   cmMendrelCathodeFrontClamp.configuration.disableFeedbackHomePos := FALSE;
   cmMendrelCathodeFrontClamp.configuration.disableFeedbackWorkPos := FALSE;
   cmMendrelCathodeFrontClamp.configuration.disableAlarms := FALSE;
   cmMendrelCathodeFrontClamp.configuration.resetOutputsOnError := FALSE;
   cmMendrelCathodeFrontClamp.configuration.allwaysWaitOnReachingTime := FALSE;
   cmMendrelCathodeRearClamp.commands.refreshConfiguration := FALSE;
   cmMendrelCathodeRearClamp.commands.editConfiguration := FALSE;
   cmMendrelCathodeRearClamp.commands.saveConfiguration := FALSE;
   cmMendrelCathodeRearClamp.commands.reset := FALSE;
   cmMendrelCathodeRearClamp.commands.commandHomePos := FALSE;
   cmMendrelCathodeRearClamp.commands.commandWorkPos := FALSE;
   cmMendrelCathodeRearClamp.monitoring.enable := TRUE;
   cmMendrelCathodeRearClamp.monitoring.referenceDesignator := WSTRING#'MendrelCathodeRearClamp';
   cmMendrelCathodeRearClamp.monitoring.commandHomePos := FALSE;
   cmMendrelCathodeRearClamp.monitoring.commandWorkPos := FALSE;
   cmMendrelCathodeRearClamp.monitoring.goToHomePos := FALSE;
   cmMendrelCathodeRearClamp.monitoring.goToWorkPos := TRUE;
   cmMendrelCathodeRearClamp.monitoring.inHomePos := FALSE;
   cmMendrelCathodeRearClamp.monitoring.inWorkPos := TRUE;
   cmMendrelCathodeRearClamp.monitoring.reset := FALSE;
   cmMendrelCathodeRearClamp.monitoring.enableManualCmds := FALSE;
   cmMendrelCathodeRearClamp.monitoring.error := FALSE;
   cmMendrelCathodeRearClamp.monitoring.interlockHomePos := TRUE;
   cmMendrelCathodeRearClamp.monitoring.interlockWorkPos := TRUE;
   cmMendrelCathodeRearClamp.monitoring.status := 16#7006;
   cmMendrelCathodeRearClamp.monitoring.interlockWarningWorkPos := FALSE;
   cmMendrelCathodeRearClamp.monitoring.interlockWarningHomePos := FALSE;
   cmMendrelCathodeRearClamp.configuration.referenceDesignator := WSTRING#'TwoWayAct.';
   cmMendrelCathodeRearClamp.configuration.monitoringLeavingFeedback := T#5S;
   cmMendrelCathodeRearClamp.configuration.monitoringReachingFeedback := T#5S;
   cmMendrelCathodeRearClamp.configuration.monitoringDiscrepancy := T#0MS;
   cmMendrelCathodeRearClamp.configuration.setOutputHomeContinuously := TRUE;
   cmMendrelCathodeRearClamp.configuration.setOutputWorkContinuously := TRUE;
   cmMendrelCathodeRearClamp.configuration.disableHomeCommand := FALSE;
   cmMendrelCathodeRearClamp.configuration.disableFeedbackHomePos := FALSE;
   cmMendrelCathodeRearClamp.configuration.disableFeedbackWorkPos := FALSE;
   cmMendrelCathodeRearClamp.configuration.disableAlarms := FALSE;
   cmMendrelCathodeRearClamp.configuration.resetOutputsOnError := FALSE;
   cmMendrelCathodeRearClamp.configuration.allwaysWaitOnReachingTime := FALSE;
   cmStackTableVaccum.commands.refreshConfiguration := FALSE;
   cmStackTableVaccum.commands.editConfiguration := FALSE;
   cmStackTableVaccum.commands.saveConfiguration := FALSE;
   cmStackTableVaccum.commands.reset := FALSE;
   cmStackTableVaccum.commands.commandHomePos := FALSE;
   cmStackTableVaccum.commands.commandWorkPos := FALSE;
   cmStackTableVaccum.monitoring.enable := TRUE;
   cmStackTableVaccum.monitoring.referenceDesignator := WSTRING#'StackTableVaccum';
   cmStackTableVaccum.monitoring.commandHomePos := FALSE;
   cmStackTableVaccum.monitoring.commandWorkPos := FALSE;
   cmStackTableVaccum.monitoring.goToHomePos := FALSE;
   cmStackTableVaccum.monitoring.goToWorkPos := FALSE;
   cmStackTableVaccum.monitoring.inHomePos := TRUE;
   cmStackTableVaccum.monitoring.inWorkPos := FALSE;
   cmStackTableVaccum.monitoring.reset := FALSE;
   cmStackTableVaccum.monitoring.enableManualCmds := FALSE;
   cmStackTableVaccum.monitoring.error := FALSE;
   cmStackTableVaccum.monitoring.interlockHomePos := TRUE;
   cmStackTableVaccum.monitoring.interlockWorkPos := TRUE;
   cmStackTableVaccum.monitoring.status := 16#7003;
   cmStackTableVaccum.monitoring.interlockWarningWorkPos := FALSE;
   cmStackTableVaccum.monitoring.interlockWarningHomePos := FALSE;
   cmStackTableVaccum.configuration.referenceDesignator := WSTRING#'TwoWayAct.';
   cmStackTableVaccum.configuration.monitoringLeavingFeedback := T#5S;
   cmStackTableVaccum.configuration.monitoringReachingFeedback := T#5S;
   cmStackTableVaccum.configuration.monitoringDiscrepancy := T#0MS;
   cmStackTableVaccum.configuration.setOutputHomeContinuously := TRUE;
   cmStackTableVaccum.configuration.setOutputWorkContinuously := TRUE;
   cmStackTableVaccum.configuration.disableHomeCommand := FALSE;
   cmStackTableVaccum.configuration.disableFeedbackHomePos := FALSE;
   cmStackTableVaccum.configuration.disableFeedbackWorkPos := FALSE;
   cmStackTableVaccum.configuration.disableAlarms := FALSE;
   cmStackTableVaccum.configuration.resetOutputsOnError := FALSE;
   cmStackTableVaccum.configuration.allwaysWaitOnReachingTime := FALSE;
   cmStackTableGapPadUpDown.commands.refreshConfiguration := FALSE;
   cmStackTableGapPadUpDown.commands.editConfiguration := FALSE;
   cmStackTableGapPadUpDown.commands.saveConfiguration := FALSE;
   cmStackTableGapPadUpDown.commands.reset := FALSE;
   cmStackTableGapPadUpDown.commands.commandHomePos := FALSE;
   cmStackTableGapPadUpDown.commands.commandWorkPos := FALSE;
   cmStackTableGapPadUpDown.monitoring.enable := TRUE;
   cmStackTableGapPadUpDown.monitoring.referenceDesignator := WSTRING#'StackTableGapPadUpDown';
   cmStackTableGapPadUpDown.monitoring.commandHomePos := FALSE;
   cmStackTableGapPadUpDown.monitoring.commandWorkPos := FALSE;
   cmStackTableGapPadUpDown.monitoring.goToHomePos := TRUE;
   cmStackTableGapPadUpDown.monitoring.goToWorkPos := FALSE;
   cmStackTableGapPadUpDown.monitoring.inHomePos := TRUE;
   cmStackTableGapPadUpDown.monitoring.inWorkPos := FALSE;
   cmStackTableGapPadUpDown.monitoring.reset := FALSE;
   cmStackTableGapPadUpDown.monitoring.enableManualCmds := FALSE;
   cmStackTableGapPadUpDown.monitoring.error := FALSE;
   cmStackTableGapPadUpDown.monitoring.interlockHomePos := TRUE;
   cmStackTableGapPadUpDown.monitoring.interlockWorkPos := TRUE;
   cmStackTableGapPadUpDown.monitoring.status := 16#7004;
   cmStackTableGapPadUpDown.monitoring.interlockWarningWorkPos := FALSE;
   cmStackTableGapPadUpDown.monitoring.interlockWarningHomePos := FALSE;
   cmStackTableGapPadUpDown.configuration.referenceDesignator := WSTRING#'TwoWayAct.';
   cmStackTableGapPadUpDown.configuration.monitoringLeavingFeedback := T#5S;
   cmStackTableGapPadUpDown.configuration.monitoringReachingFeedback := T#5S;
   cmStackTableGapPadUpDown.configuration.monitoringDiscrepancy := T#0MS;
   cmStackTableGapPadUpDown.configuration.setOutputHomeContinuously := TRUE;
   cmStackTableGapPadUpDown.configuration.setOutputWorkContinuously := TRUE;
   cmStackTableGapPadUpDown.configuration.disableHomeCommand := FALSE;
   cmStackTableGapPadUpDown.configuration.disableFeedbackHomePos := FALSE;
   cmStackTableGapPadUpDown.configuration.disableFeedbackWorkPos := FALSE;
   cmStackTableGapPadUpDown.configuration.disableAlarms := FALSE;
   cmStackTableGapPadUpDown.configuration.resetOutputsOnError := FALSE;
   cmStackTableGapPadUpDown.configuration.allwaysWaitOnReachingTime := FALSE;
   cmStackTableVisionControllerInterface.commands.stepStart := FALSE;
   cmStackTableVisionControllerInterface.commands.errorAck := FALSE;
   cmStackTableVisionControllerInterface.commands.dataDelete := FALSE;
   cmStackTableVisionControllerInterface.monitoring.profinetInput.cmdResultStatus.cmdComplete := FALSE;
   cmStackTableVisionControllerInterface.monitoring.profinetInput.cmdResultStatus.cmdError := FALSE;
   cmStackTableVisionControllerInterface.monitoring.profinetInput.cmdResultStatus.cmdReady := FALSE;
   cmStackTableVisionControllerInterface.monitoring.profinetInput.cmdResultStatus.resultReady := FALSE;
   cmStackTableVisionControllerInterface.monitoring.profinetInput.cmdResultStatus.resultOR := FALSE;
   cmStackTableVisionControllerInterface.monitoring.profinetInput.cmdResultStatus.reserved0 := FALSE;
   cmStackTableVisionControllerInterface.monitoring.profinetInput.cmdResultStatus.reserved1 := FALSE;
   cmStackTableVisionControllerInterface.monitoring.profinetInput.cmdResultStatus.reserved2 := FALSE;
   cmStackTableVisionControllerInterface.monitoring.profinetInput.trgReadyStatus.trg1Ready := FALSE;
   cmStackTableVisionControllerInterface.monitoring.profinetInput.trgReadyStatus.trg2Ready := FALSE;
   cmStackTableVisionControllerInterface.monitoring.profinetInput.trgReadyStatus.trg3Ready := FALSE;
   cmStackTableVisionControllerInterface.monitoring.profinetInput.trgReadyStatus.trg4Ready := FALSE;
   cmStackTableVisionControllerInterface.monitoring.profinetInput.trgReadyStatus.reserved0 := FALSE;
   cmStackTableVisionControllerInterface.monitoring.profinetInput.trgReadyStatus.reserved1 := FALSE;
   cmStackTableVisionControllerInterface.monitoring.profinetInput.trgReadyStatus.reserved2 := FALSE;
   cmStackTableVisionControllerInterface.monitoring.profinetInput.trgReadyStatus.reserved3 := FALSE;
   cmStackTableVisionControllerInterface.monitoring.profinetInput.trgAckStatus.trg1Ack := FALSE;
   cmStackTableVisionControllerInterface.monitoring.profinetInput.trgAckStatus.trg2Ack := FALSE;
   cmStackTableVisionControllerInterface.monitoring.profinetInput.trgAckStatus.trg3Ack := FALSE;
   cmStackTableVisionControllerInterface.monitoring.profinetInput.trgAckStatus.trg4Ack := FALSE;
   cmStackTableVisionControllerInterface.monitoring.profinetInput.trgAckStatus.reserved0 := FALSE;
   cmStackTableVisionControllerInterface.monitoring.profinetInput.trgAckStatus.reserved1 := FALSE;
   cmStackTableVisionControllerInterface.monitoring.profinetInput.trgAckStatus.reserved2 := FALSE;
   cmStackTableVisionControllerInterface.monitoring.profinetInput.trgAckStatus.reserved3 := FALSE;
   cmStackTableVisionControllerInterface.monitoring.profinetInput.miscellaneousStatus.busy := FALSE;
   cmStackTableVisionControllerInterface.monitoring.profinetInput.miscellaneousStatus.err0Status := FALSE;
   cmStackTableVisionControllerInterface.monitoring.profinetInput.miscellaneousStatus.err1Status := FALSE;
   cmStackTableVisionControllerInterface.monitoring.profinetInput.miscellaneousStatus.remoteReady := FALSE;
   cmStackTableVisionControllerInterface.monitoring.profinetInput.miscellaneousStatus.reserved0 := FALSE;
   cmStackTableVisionControllerInterface.monitoring.profinetInput.miscellaneousStatus.reserved1 := FALSE;
   cmStackTableVisionControllerInterface.monitoring.profinetInput.miscellaneousStatus.reserved2 := FALSE;
   cmStackTableVisionControllerInterface.monitoring.profinetInput.miscellaneousStatus.reserved3 := FALSE;
   cmStackTableVisionControllerInterface.monitoring.profinetInput.assignableStatus.assignable_0 := FALSE;
   cmStackTableVisionControllerInterface.monitoring.profinetInput.assignableStatus.assignable_1 := FALSE;
   cmStackTableVisionControllerInterface.monitoring.profinetInput.assignableStatus.assignable_2 := FALSE;
   cmStackTableVisionControllerInterface.monitoring.profinetInput.assignableStatus.assignable_3 := FALSE;
   cmStackTableVisionControllerInterface.monitoring.profinetInput.assignableStatus.assignable_4 := FALSE;
   cmStackTableVisionControllerInterface.monitoring.profinetInput.assignableStatus.assignable_5 := FALSE;
   cmStackTableVisionControllerInterface.monitoring.profinetInput.assignableStatus.assignable_6 := FALSE;
   cmStackTableVisionControllerInterface.monitoring.profinetInput.assignableStatus.assignable_7 := FALSE;
   cmStackTableVisionControllerInterface.monitoring.profinetInput.assignableStatus.assignable_8 := FALSE;
   cmStackTableVisionControllerInterface.monitoring.profinetInput.assignableStatus.assignable_9 := FALSE;
   cmStackTableVisionControllerInterface.monitoring.profinetInput.assignableStatus.assignable_10 := FALSE;
   cmStackTableVisionControllerInterface.monitoring.profinetInput.assignableStatus.assignable_11 := FALSE;
   cmStackTableVisionControllerInterface.monitoring.profinetInput.assignableStatus.assignable_12 := FALSE;
   cmStackTableVisionControllerInterface.monitoring.profinetInput.assignableStatus.assignable_13 := FALSE;
   cmStackTableVisionControllerInterface.monitoring.profinetInput.assignableStatus.assignable_14 := FALSE;
   cmStackTableVisionControllerInterface.monitoring.profinetInput.assignableStatus.assignable_15 := FALSE;
   cmStackTableVisionControllerInterface.monitoring.profinetInput.assignableStatus.assignable_16 := FALSE;
   cmStackTableVisionControllerInterface.monitoring.profinetInput.assignableStatus.assignable_17 := FALSE;
   cmStackTableVisionControllerInterface.monitoring.profinetInput.assignableStatus.assignable_18 := FALSE;
   cmStackTableVisionControllerInterface.monitoring.profinetInput.assignableStatus.assignable_19 := FALSE;
   cmStackTableVisionControllerInterface.monitoring.profinetInput.assignableStatus.assignable_20 := FALSE;
   cmStackTableVisionControllerInterface.monitoring.profinetInput.assignableStatus.assignable_21 := FALSE;
   cmStackTableVisionControllerInterface.monitoring.profinetInput.assignableStatus.assignable_22 := FALSE;
   cmStackTableVisionControllerInterface.monitoring.profinetInput.assignableStatus.assignable_23 := FALSE;
   cmStackTableVisionControllerInterface.monitoring.profinetInput.assignableStatus.assignable_24 := FALSE;
   cmStackTableVisionControllerInterface.monitoring.profinetInput.assignableStatus.assignable_25 := FALSE;
   cmStackTableVisionControllerInterface.monitoring.profinetInput.assignableStatus.assignable_26 := FALSE;
   cmStackTableVisionControllerInterface.monitoring.profinetInput.assignableStatus.assignable_27 := FALSE;
   cmStackTableVisionControllerInterface.monitoring.profinetInput.assignableStatus.assignable_28 := FALSE;
   cmStackTableVisionControllerInterface.monitoring.profinetInput.assignableStatus.assignable_29 := FALSE;
   cmStackTableVisionControllerInterface.monitoring.profinetInput.assignableStatus.assignable_30 := FALSE;
   cmStackTableVisionControllerInterface.monitoring.profinetInput.assignableStatus.assignable_31 := FALSE;
   cmStackTableVisionControllerInterface.monitoring.profinetInput.resultData248Byte_1.error0Code := 0;
   cmStackTableVisionControllerInterface.monitoring.profinetInput.resultData248Byte_1.error1Code := 0;
   cmStackTableVisionControllerInterface.monitoring.profinetInput.resultData248Byte_1.reserved12 := 0;
   cmStackTableVisionControllerInterface.monitoring.profinetInput.resultData248Byte_1.totalCount := 0;
   cmStackTableVisionControllerInterface.monitoring.profinetInput.resultData248Byte_1.commandResult := 0;
   cmStackTableVisionControllerInterface.monitoring.profinetInput.resultData248Byte_1.commandData[0..23] := 0;
   cmStackTableVisionControllerInterface.monitoring.profinetInput.resultData248Byte_1.resultData[0..33] := 0;
   cmStackTableVisionControllerInterface.monitoring.profinetInput.resultData248Byte_2[0..61] := 0;
   cmStackTableVisionControllerInterface.monitoring.profinetInput.resultData248Byte_3[0..61] := 0;
   cmStackTableVisionControllerInterface.monitoring.profinetInput.resultData248Byte_4[0..61] := 0;
   cmStackTableVisionControllerInterface.monitoring.profinetInput.resultData248Byte_5[0..61] := 0;
   cmStackTableVisionControllerInterface.monitoring.profinetOutput.cmdResultControl.cmdRequest := FALSE;
   cmStackTableVisionControllerInterface.monitoring.profinetOutput.cmdResultControl.inDataFbSyncInhibit := FALSE;
   cmStackTableVisionControllerInterface.monitoring.profinetOutput.cmdResultControl.reserved := FALSE;
   cmStackTableVisionControllerInterface.monitoring.profinetOutput.cmdResultControl.resultAck := FALSE;
   cmStackTableVisionControllerInterface.monitoring.profinetOutput.cmdResultControl.err0ResetRequest := FALSE;
   cmStackTableVisionControllerInterface.monitoring.profinetOutput.cmdResultControl.err1ResetRequest := FALSE;
   cmStackTableVisionControllerInterface.monitoring.profinetOutput.cmdResultControl.reserved0 := FALSE;
   cmStackTableVisionControllerInterface.monitoring.profinetOutput.cmdResultControl.reserved1 := FALSE;
   cmStackTableVisionControllerInterface.monitoring.profinetOutput.trgControl.trg1 := FALSE;
   cmStackTableVisionControllerInterface.monitoring.profinetOutput.trgControl.trg2 := FALSE;
   cmStackTableVisionControllerInterface.monitoring.profinetOutput.trgControl.trg3 := FALSE;
   cmStackTableVisionControllerInterface.monitoring.profinetOutput.trgControl.trg4 := FALSE;
   cmStackTableVisionControllerInterface.monitoring.profinetOutput.trgControl.reserved0 := FALSE;
   cmStackTableVisionControllerInterface.monitoring.profinetOutput.trgControl.reserved1 := FALSE;
   cmStackTableVisionControllerInterface.monitoring.profinetOutput.trgControl.reserved2 := FALSE;
   cmStackTableVisionControllerInterface.monitoring.profinetOutput.trgControl.reserved3 := FALSE;
   cmStackTableVisionControllerInterface.monitoring.profinetOutput.miscellaneousControl.reset := FALSE;
   cmStackTableVisionControllerInterface.monitoring.profinetOutput.miscellaneousControl.ext := FALSE;
   cmStackTableVisionControllerInterface.monitoring.profinetOutput.miscellaneousControl.test := FALSE;
   cmStackTableVisionControllerInterface.monitoring.profinetOutput.miscellaneousControl.reserved0 := FALSE;
   cmStackTableVisionControllerInterface.monitoring.profinetOutput.miscellaneousControl.reserved1 := FALSE;
   cmStackTableVisionControllerInterface.monitoring.profinetOutput.miscellaneousControl.reserved2 := FALSE;
   cmStackTableVisionControllerInterface.monitoring.profinetOutput.miscellaneousControl.reserved3 := FALSE;
   cmStackTableVisionControllerInterface.monitoring.profinetOutput.miscellaneousControl.reserved4 := FALSE;
   cmStackTableVisionControllerInterface.monitoring.profinetOutput.reservedControl.reserved0 := FALSE;
   cmStackTableVisionControllerInterface.monitoring.profinetOutput.reservedControl.reserved1 := FALSE;
   cmStackTableVisionControllerInterface.monitoring.profinetOutput.reservedControl.reserved2 := FALSE;
   cmStackTableVisionControllerInterface.monitoring.profinetOutput.reservedControl.reserved3 := FALSE;
   cmStackTableVisionControllerInterface.monitoring.profinetOutput.reservedControl.reserved4 := FALSE;
   cmStackTableVisionControllerInterface.monitoring.profinetOutput.reservedControl.reserved5 := FALSE;
   cmStackTableVisionControllerInterface.monitoring.profinetOutput.reservedControl.reserved6 := FALSE;
   cmStackTableVisionControllerInterface.monitoring.profinetOutput.reservedControl.reserved7 := FALSE;
   cmStackTableVisionControllerInterface.monitoring.profinetOutput.assignableControl.assignable_0 := FALSE;
   cmStackTableVisionControllerInterface.monitoring.profinetOutput.assignableControl.assignable_1 := FALSE;
   cmStackTableVisionControllerInterface.monitoring.profinetOutput.assignableControl.assignable_2 := FALSE;
   cmStackTableVisionControllerInterface.monitoring.profinetOutput.assignableControl.assignable_3 := FALSE;
   cmStackTableVisionControllerInterface.monitoring.profinetOutput.assignableControl.assignable_4 := FALSE;
   cmStackTableVisionControllerInterface.monitoring.profinetOutput.assignableControl.assignable_5 := FALSE;
   cmStackTableVisionControllerInterface.monitoring.profinetOutput.assignableControl.assignable_6 := FALSE;
   cmStackTableVisionControllerInterface.monitoring.profinetOutput.assignableControl.assignable_7 := FALSE;
   cmStackTableVisionControllerInterface.monitoring.profinetOutput.assignableControl.assignable_8 := FALSE;
   cmStackTableVisionControllerInterface.monitoring.profinetOutput.assignableControl.assignable_9 := FALSE;
   cmStackTableVisionControllerInterface.monitoring.profinetOutput.assignableControl.assignable_10 := FALSE;
   cmStackTableVisionControllerInterface.monitoring.profinetOutput.assignableControl.assignable_11 := FALSE;
   cmStackTableVisionControllerInterface.monitoring.profinetOutput.assignableControl.assignable_12 := FALSE;
   cmStackTableVisionControllerInterface.monitoring.profinetOutput.assignableControl.assignable_13 := FALSE;
   cmStackTableVisionControllerInterface.monitoring.profinetOutput.assignableControl.assignable_14 := FALSE;
   cmStackTableVisionControllerInterface.monitoring.profinetOutput.assignableControl.assignable_15 := FALSE;
   cmStackTableVisionControllerInterface.monitoring.profinetOutput.assignableControl.assignable_16 := FALSE;
   cmStackTableVisionControllerInterface.monitoring.profinetOutput.assignableControl.assignable_17 := FALSE;
   cmStackTableVisionControllerInterface.monitoring.profinetOutput.assignableControl.assignable_18 := FALSE;
   cmStackTableVisionControllerInterface.monitoring.profinetOutput.assignableControl.assignable_19 := FALSE;
   cmStackTableVisionControllerInterface.monitoring.profinetOutput.assignableControl.assignable_20 := FALSE;
   cmStackTableVisionControllerInterface.monitoring.profinetOutput.assignableControl.assignable_21 := FALSE;
   cmStackTableVisionControllerInterface.monitoring.profinetOutput.assignableControl.assignable_22 := FALSE;
   cmStackTableVisionControllerInterface.monitoring.profinetOutput.assignableControl.assignable_23 := FALSE;
   cmStackTableVisionControllerInterface.monitoring.profinetOutput.assignableControl.assignable_24 := FALSE;
   cmStackTableVisionControllerInterface.monitoring.profinetOutput.assignableControl.assignable_25 := FALSE;
   cmStackTableVisionControllerInterface.monitoring.profinetOutput.assignableControl.assignable_26 := FALSE;
   cmStackTableVisionControllerInterface.monitoring.profinetOutput.assignableControl.assignable_27 := FALSE;
   cmStackTableVisionControllerInterface.monitoring.profinetOutput.assignableControl.assignable_28 := FALSE;
   cmStackTableVisionControllerInterface.monitoring.profinetOutput.assignableControl.assignable_29 := FALSE;
   cmStackTableVisionControllerInterface.monitoring.profinetOutput.assignableControl.assignable_30 := FALSE;
   cmStackTableVisionControllerInterface.monitoring.profinetOutput.assignableControl.assignable_31 := FALSE;
   cmStackTableVisionControllerInterface.monitoring.profinetOutput.parameterData248Byte_1.reversed0 := 0;
   cmStackTableVisionControllerInterface.monitoring.profinetOutput.parameterData248Byte_1.reserved1 := 0;
   cmStackTableVisionControllerInterface.monitoring.profinetOutput.parameterData248Byte_1.commandNumber := 0;
   cmStackTableVisionControllerInterface.monitoring.profinetOutput.parameterData248Byte_1.cmdParameter[0..15] := 0;
   cmStackTableVisionControllerInterface.monitoring.profinetOutput.parameterData248Byte_1.inDataFieldbus[0..42] := 0;
   cmStackTableVisionControllerInterface.monitoring.profinetOutput.parameterData248Byte_2[0..61] := 0;
   cmStackTableVisionControllerInterface.monitoring.profinetOutput.parameterData248Byte_3[0..61] := 0;
   cmStackTableVisionControllerInterface.monitoring.profinetOutput.parameterData248Byte_4[0..61] := 0;
   cmStackTableVisionControllerInterface.monitoring.profinetOutput.parameterData248Byte_5[0..61] := 0;
   cmStackTableVisionControllerInterface.monitoring.resultOK := FALSE;
   cmStackTableVisionControllerInterface.monitoring.resultNG := FALSE;
   cmStackTableVisionControllerInterface.monitoring.resultBusy := FALSE;
   cmStackTableVisionControllerInterface.monitoring.resultComplete := FALSE;
   cmStackTableVisionControllerInterface.monitoring.resultData.resultData136Byte_1[0..33] := 0;
   cmStackTableVisionControllerInterface.monitoring.resultData.resultData248Byte_2[0..61] := 0;
   cmStackTableVisionControllerInterface.monitoring.resultData.resultData248Byte_3[0..61] := 0;
   cmStackTableVisionControllerInterface.monitoring.resultData.resultData248Byte_4[0..61] := 0;
   cmStackTableVisionControllerInterface.monitoring.resultData.resultData248Byte_5[0..61] := 0;
   cmStackTableVisionControllerInterface.monitoring.error := FALSE;
   cmStackTableVisionControllerInterface.monitoring.status := 16#0000;
   cmStackTableVisionControllerInterface.configuration.hwID.cmdResultStatusID := 0;
   cmStackTableVisionControllerInterface.configuration.hwID.trgReadyStatusID := 0;
   cmStackTableVisionControllerInterface.configuration.hwID.trgAckStatusID := 0;
   cmStackTableVisionControllerInterface.configuration.hwID.miscellaneousStatusID := 0;
   cmStackTableVisionControllerInterface.configuration.hwID.assignableStatusID := 0;
   cmStackTableVisionControllerInterface.configuration.hwID.resultData248ByteID_1 := 0;
   cmStackTableVisionControllerInterface.configuration.hwID.resultData248ByteID_2 := 0;
   cmStackTableVisionControllerInterface.configuration.hwID.resultData248ByteID_3 := 0;
   cmStackTableVisionControllerInterface.configuration.hwID.resultData248ByteID_4 := 0;
   cmStackTableVisionControllerInterface.configuration.hwID.resultData248ByteID_5 := 0;
   cmStackTableVisionControllerInterface.configuration.hwID.cmdResultControlID := 0;
   cmStackTableVisionControllerInterface.configuration.hwID.trgControlID := 0;
   cmStackTableVisionControllerInterface.configuration.hwID.miscellaneousControlID := 0;
   cmStackTableVisionControllerInterface.configuration.hwID.reservedControlID := 0;
   cmStackTableVisionControllerInterface.configuration.hwID.assignableControlID := 0;
   cmStackTableVisionControllerInterface.configuration.hwID.parameterData248ByteID_1 := 0;
   cmStackTableVisionControllerInterface.configuration.hwID.parameterData248ByteID_2 := 0;
   cmStackTableVisionControllerInterface.configuration.hwID.parameterData248ByteID_3 := 0;
   cmStackTableVisionControllerInterface.configuration.hwID.parameterData248ByteID_4 := 0;
   cmStackTableVisionControllerInterface.configuration.hwID.parameterData248ByteID_5 := 0;
   cmStackTableVisionControllerInterface.configuration.referenceDesignator := WSTRING#'';
   cmStackTableVisionControllerInterface.configuration.disableAlarms := FALSE;
   cmStackTableVisionControllerInterface.configuration.trigger1Use := FALSE;
   cmStackTableVisionControllerInterface.configuration.trigger2Use := FALSE;
   cmStackTableVisionControllerInterface.configuration.trigger3Use := FALSE;
   cmStackTableVisionControllerInterface.configuration.trigger4Use := FALSE;
   cmStackTableVisionControllerInterface.configuration.triggertime := T#0MS;
   cmStackTableVisionControllerInterface.configuration.cycleTime := T#0MS;
   cmStackTableVisionControllerInterface.configuration.DataConfig.cmdResultControl.cmdRequest := FALSE;
   cmStackTableVisionControllerInterface.configuration.DataConfig.cmdResultControl.inDataFbSyncInhibit := FALSE;
   cmStackTableVisionControllerInterface.configuration.DataConfig.cmdResultControl.reserved := FALSE;
   cmStackTableVisionControllerInterface.configuration.DataConfig.cmdResultControl.resultAck := FALSE;
   cmStackTableVisionControllerInterface.configuration.DataConfig.cmdResultControl.err0ResetRequest := FALSE;
   cmStackTableVisionControllerInterface.configuration.DataConfig.cmdResultControl.err1ResetRequest := FALSE;
   cmStackTableVisionControllerInterface.configuration.DataConfig.cmdResultControl.reserved0 := FALSE;
   cmStackTableVisionControllerInterface.configuration.DataConfig.cmdResultControl.reserved1 := FALSE;
   cmStackTableVisionControllerInterface.configuration.DataConfig.trgControl.trg1 := FALSE;
   cmStackTableVisionControllerInterface.configuration.DataConfig.trgControl.trg2 := FALSE;
   cmStackTableVisionControllerInterface.configuration.DataConfig.trgControl.trg3 := FALSE;
   cmStackTableVisionControllerInterface.configuration.DataConfig.trgControl.trg4 := FALSE;
   cmStackTableVisionControllerInterface.configuration.DataConfig.trgControl.reserved0 := FALSE;
   cmStackTableVisionControllerInterface.configuration.DataConfig.trgControl.reserved1 := FALSE;
   cmStackTableVisionControllerInterface.configuration.DataConfig.trgControl.reserved2 := FALSE;
   cmStackTableVisionControllerInterface.configuration.DataConfig.trgControl.reserved3 := FALSE;
   cmStackTableVisionControllerInterface.configuration.DataConfig.miscellaneousControl.reset := FALSE;
   cmStackTableVisionControllerInterface.configuration.DataConfig.miscellaneousControl.ext := FALSE;
   cmStackTableVisionControllerInterface.configuration.DataConfig.miscellaneousControl.test := FALSE;
   cmStackTableVisionControllerInterface.configuration.DataConfig.miscellaneousControl.reserved0 := FALSE;
   cmStackTableVisionControllerInterface.configuration.DataConfig.miscellaneousControl.reserved1 := FALSE;
   cmStackTableVisionControllerInterface.configuration.DataConfig.miscellaneousControl.reserved2 := FALSE;
   cmStackTableVisionControllerInterface.configuration.DataConfig.miscellaneousControl.reserved3 := FALSE;
   cmStackTableVisionControllerInterface.configuration.DataConfig.miscellaneousControl.reserved4 := FALSE;
   cmStackTableVisionControllerInterface.configuration.DataConfig.reservedControl.reserved0 := FALSE;
   cmStackTableVisionControllerInterface.configuration.DataConfig.reservedControl.reserved1 := FALSE;
   cmStackTableVisionControllerInterface.configuration.DataConfig.reservedControl.reserved2 := FALSE;
   cmStackTableVisionControllerInterface.configuration.DataConfig.reservedControl.reserved3 := FALSE;
   cmStackTableVisionControllerInterface.configuration.DataConfig.reservedControl.reserved4 := FALSE;
   cmStackTableVisionControllerInterface.configuration.DataConfig.reservedControl.reserved5 := FALSE;
   cmStackTableVisionControllerInterface.configuration.DataConfig.reservedControl.reserved6 := FALSE;
   cmStackTableVisionControllerInterface.configuration.DataConfig.reservedControl.reserved7 := FALSE;
   cmStackTableVisionControllerInterface.configuration.DataConfig.assignableControl.assignable_0 := FALSE;
   cmStackTableVisionControllerInterface.configuration.DataConfig.assignableControl.assignable_1 := FALSE;
   cmStackTableVisionControllerInterface.configuration.DataConfig.assignableControl.assignable_2 := FALSE;
   cmStackTableVisionControllerInterface.configuration.DataConfig.assignableControl.assignable_3 := FALSE;
   cmStackTableVisionControllerInterface.configuration.DataConfig.assignableControl.assignable_4 := FALSE;
   cmStackTableVisionControllerInterface.configuration.DataConfig.assignableControl.assignable_5 := FALSE;
   cmStackTableVisionControllerInterface.configuration.DataConfig.assignableControl.assignable_6 := FALSE;
   cmStackTableVisionControllerInterface.configuration.DataConfig.assignableControl.assignable_7 := FALSE;
   cmStackTableVisionControllerInterface.configuration.DataConfig.assignableControl.assignable_8 := FALSE;
   cmStackTableVisionControllerInterface.configuration.DataConfig.assignableControl.assignable_9 := FALSE;
   cmStackTableVisionControllerInterface.configuration.DataConfig.assignableControl.assignable_10 := FALSE;
   cmStackTableVisionControllerInterface.configuration.DataConfig.assignableControl.assignable_11 := FALSE;
   cmStackTableVisionControllerInterface.configuration.DataConfig.assignableControl.assignable_12 := FALSE;
   cmStackTableVisionControllerInterface.configuration.DataConfig.assignableControl.assignable_13 := FALSE;
   cmStackTableVisionControllerInterface.configuration.DataConfig.assignableControl.assignable_14 := FALSE;
   cmStackTableVisionControllerInterface.configuration.DataConfig.assignableControl.assignable_15 := FALSE;
   cmStackTableVisionControllerInterface.configuration.DataConfig.assignableControl.assignable_16 := FALSE;
   cmStackTableVisionControllerInterface.configuration.DataConfig.assignableControl.assignable_17 := FALSE;
   cmStackTableVisionControllerInterface.configuration.DataConfig.assignableControl.assignable_18 := FALSE;
   cmStackTableVisionControllerInterface.configuration.DataConfig.assignableControl.assignable_19 := FALSE;
   cmStackTableVisionControllerInterface.configuration.DataConfig.assignableControl.assignable_20 := FALSE;
   cmStackTableVisionControllerInterface.configuration.DataConfig.assignableControl.assignable_21 := FALSE;
   cmStackTableVisionControllerInterface.configuration.DataConfig.assignableControl.assignable_22 := FALSE;
   cmStackTableVisionControllerInterface.configuration.DataConfig.assignableControl.assignable_23 := FALSE;
   cmStackTableVisionControllerInterface.configuration.DataConfig.assignableControl.assignable_24 := FALSE;
   cmStackTableVisionControllerInterface.configuration.DataConfig.assignableControl.assignable_25 := FALSE;
   cmStackTableVisionControllerInterface.configuration.DataConfig.assignableControl.assignable_26 := FALSE;
   cmStackTableVisionControllerInterface.configuration.DataConfig.assignableControl.assignable_27 := FALSE;
   cmStackTableVisionControllerInterface.configuration.DataConfig.assignableControl.assignable_28 := FALSE;
   cmStackTableVisionControllerInterface.configuration.DataConfig.assignableControl.assignable_29 := FALSE;
   cmStackTableVisionControllerInterface.configuration.DataConfig.assignableControl.assignable_30 := FALSE;
   cmStackTableVisionControllerInterface.configuration.DataConfig.assignableControl.assignable_31 := FALSE;
   cmStackTableVisionControllerInterface.configuration.DataConfig.parameterData248Byte_1.reversed0 := 0;
   cmStackTableVisionControllerInterface.configuration.DataConfig.parameterData248Byte_1.reserved1 := 0;
   cmStackTableVisionControllerInterface.configuration.DataConfig.parameterData248Byte_1.commandNumber := 0;
   cmStackTableVisionControllerInterface.configuration.DataConfig.parameterData248Byte_1.cmdParameter[0..15] := 0;
   cmStackTableVisionControllerInterface.configuration.DataConfig.parameterData248Byte_1.inDataFieldbus[0..42] := 0;
   cmStackTableVisionControllerInterface.configuration.DataConfig.parameterData248Byte_2[0..61] := 0;
   cmStackTableVisionControllerInterface.configuration.DataConfig.parameterData248Byte_3[0..61] := 0;
   cmStackTableVisionControllerInterface.configuration.DataConfig.parameterData248Byte_4[0..61] := 0;
   cmStackTableVisionControllerInterface.configuration.DataConfig.parameterData248Byte_5[0..61] := 0;
   StackTableVisionHistory.partID[0..50] := '';
   StackTableVisionHistory.productionTimestamp[0..50] := DTL#1970-01-01-00:00:00;
   StackTableVisionHistory.data[0..50].VisionOk := FALSE;
   StackTableVisionHistory.data[0..50].VisionNG := FALSE;
   StackTableVisionHistory.data[0..50].VisionComplete := FALSE;
   StackTableVisionHistory.data[0..50]."GagueR&Rtype1OK" := FALSE;
   StackTableVisionHistory.data[0..50]."GagueR&Rtype1NG" := FALSE;
   StackTableVisionHistory.data[0..50]."GagueR&Rtype1Complete" := FALSE;
   StackTableVisionHistory.data[0..50]."GagueR&Rtype3OK" := FALSE;
   StackTableVisionHistory.data[0..50]."GagueR&Rtype3NG" := FALSE;
   StackTableVisionHistory.data[0..50]."GagueR&Rtype3Complete" := FALSE;
   StackTableVisionHistory.data[0..50].VisionData.tabFoldingMissingJudgementResult := 0.0;
   StackTableVisionHistory.data[0..50].VisionData.electrodeLengthJudgementResult := 0.0;
   StackTableVisionHistory.data[0..50].VisionData.electrodeHeightJudgementResult := 0.0;
   StackTableVisionHistory.data[0..50].VisionData.movementAmountAxisX1 := 0.0;
   StackTableVisionHistory.data[0..50].VisionData.movementAmountAxisY1 := 0.0;
   StackTableVisionHistory.data[0..50].VisionData.movementAmountAxisY2 := 0.0;
   StackTableVisionHistory.data[0..50].VisionData.tabFoldingMissingReply := 0.0;
   StackTableVisionHistory.data[0..50].VisionData.tabFoldingMissingUpperRangeReply := 0.0;
   StackTableVisionHistory.data[0..50].VisionData.tabFoldingMissingLowerRangeReply := 0.0;
   StackTableVisionHistory.data[0..50].VisionData.electrodeLengthReply := 0.0;
   StackTableVisionHistory.data[0..50].VisionData.electrodeLengthUpperRangeReply := 0.0;
   StackTableVisionHistory.data[0..50].VisionData.electrodeLengthLowerRangeReply := 0.0;
   StackTableVisionHistory.data[0..50].VisionData.electrodeHeightReply := 0.0;
   StackTableVisionHistory.data[0..50].VisionData.electrodeHeightUpperRangeReply := 0.0;
   StackTableVisionHistory.data[0..50].VisionData.electrodeHeightLowerRangeReply := 0.0;
   intCondition.Axis_21.Home.HomeInterlock := FALSE;
   intCondition.Axis_21.Home.homeinterlock_error := FALSE;
   intCondition.Axis_21.Home.intout[0..9] := FALSE;
   intCondition.Axis_21.Jog.ForwardInterlockOK := FALSE;
   intCondition.Axis_21.Jog.BackwardInterlockOk := FALSE;
   intCondition.Axis_21.Jog.ForwardInterlockError := FALSE;
   intCondition.Axis_21.Jog.BackwardInterlockError := FALSE;
   intCondition.Axis_21.Jog.intOut[0..9] := FALSE;
   intCondition.Axis_21.Position.interlockOk[0..15] := FALSE;
   intCondition.Axis_21.Position.interlockError[0..15] := FALSE;
   intCondition.Axis_21.Position.intOut[0..9] := FALSE;
   intCondition.Axis_22.Home.HomeInterlock := FALSE;
   intCondition.Axis_22.Home.homeinterlock_error := FALSE;
   intCondition.Axis_22.Home.intout[0..9] := FALSE;
   intCondition.Axis_22.Jog.ForwardInterlockOK := FALSE;
   intCondition.Axis_22.Jog.BackwardInterlockOk := FALSE;
   intCondition.Axis_22.Jog.ForwardInterlockError := FALSE;
   intCondition.Axis_22.Jog.BackwardInterlockError := FALSE;
   intCondition.Axis_22.Jog.intOut[0..9] := FALSE;
   intCondition.Axis_22.Position.interlockOk[0..15] := FALSE;
   intCondition.Axis_22.Position.interlockError[0..15] := FALSE;
   intCondition.Axis_22.Position.intOut[0..9] := FALSE;
   intCondition.Axis_23.Home.HomeInterlock := FALSE;
   intCondition.Axis_23.Home.homeinterlock_error := FALSE;
   intCondition.Axis_23.Home.intout[0..9] := FALSE;
   intCondition.Axis_23.Jog.ForwardInterlockOK := FALSE;
   intCondition.Axis_23.Jog.BackwardInterlockOk := FALSE;
   intCondition.Axis_23.Jog.ForwardInterlockError := FALSE;
   intCondition.Axis_23.Jog.BackwardInterlockError := FALSE;
   intCondition.Axis_23.Jog.intOut[0..9] := FALSE;
   intCondition.Axis_23.Position.interlockOk[0..15] := FALSE;
   intCondition.Axis_23.Position.interlockError[0..15] := FALSE;
   intCondition.Axis_23.Position.intOut[0..9] := FALSE;
   intCondition.Axis_24.Home.HomeInterlock := FALSE;
   intCondition.Axis_24.Home.homeinterlock_error := FALSE;
   intCondition.Axis_24.Home.intout[0..9] := FALSE;
   intCondition.Axis_24.Jog.ForwardInterlockOK := FALSE;
   intCondition.Axis_24.Jog.BackwardInterlockOk := FALSE;
   intCondition.Axis_24.Jog.ForwardInterlockError := FALSE;
   intCondition.Axis_24.Jog.BackwardInterlockError := FALSE;
   intCondition.Axis_24.Jog.intOut[0..9] := FALSE;
   intCondition.Axis_24.Position.interlockOk[0..15] := FALSE;
   intCondition.Axis_24.Position.interlockError[0..15] := FALSE;
   intCondition.Axis_24.Position.intOut[0..9] := FALSE;
   intCondition.Axis_25.Home.HomeInterlock := FALSE;
   intCondition.Axis_25.Home.homeinterlock_error := FALSE;
   intCondition.Axis_25.Home.intout[0..9] := FALSE;
   intCondition.Axis_25.Jog.ForwardInterlockOK := FALSE;
   intCondition.Axis_25.Jog.BackwardInterlockOk := FALSE;
   intCondition.Axis_25.Jog.ForwardInterlockError := FALSE;
   intCondition.Axis_25.Jog.BackwardInterlockError := FALSE;
   intCondition.Axis_25.Jog.intOut[0..9] := FALSE;
   intCondition.Axis_25.Position.interlockOk[0..15] := FALSE;
   intCondition.Axis_25.Position.interlockError[0..15] := FALSE;
   intCondition.Axis_25.Position.intOut[0..9] := FALSE;
   intCondition.Axis_26.Home.HomeInterlock := FALSE;
   intCondition.Axis_26.Home.homeinterlock_error := FALSE;
   intCondition.Axis_26.Home.intout[0..9] := FALSE;
   intCondition.Axis_26.Jog.ForwardInterlockOK := FALSE;
   intCondition.Axis_26.Jog.BackwardInterlockOk := FALSE;
   intCondition.Axis_26.Jog.ForwardInterlockError := FALSE;
   intCondition.Axis_26.Jog.BackwardInterlockError := FALSE;
   intCondition.Axis_26.Jog.intOut[0..9] := FALSE;
   intCondition.Axis_26.Position.interlockOk[0..15] := FALSE;
   intCondition.Axis_26.Position.interlockError[0..15] := FALSE;
   intCondition.Axis_26.Position.intOut[0..9] := FALSE;
   intCondition.Axis_27.Home.HomeInterlock := FALSE;
   intCondition.Axis_27.Home.homeinterlock_error := FALSE;
   intCondition.Axis_27.Home.intout[0..9] := FALSE;
   intCondition.Axis_27.Jog.ForwardInterlockOK := FALSE;
   intCondition.Axis_27.Jog.BackwardInterlockOk := FALSE;
   intCondition.Axis_27.Jog.ForwardInterlockError := FALSE;
   intCondition.Axis_27.Jog.BackwardInterlockError := FALSE;
   intCondition.Axis_27.Jog.intOut[0..9] := FALSE;
   intCondition.Axis_27.Position.interlockOk[0..15] := FALSE;
   intCondition.Axis_27.Position.interlockError[0..15] := FALSE;
   intCondition.Axis_27.Position.intOut[0..9] := FALSE;
   intCondition.Axis_28.Home.HomeInterlock := FALSE;
   intCondition.Axis_28.Home.homeinterlock_error := FALSE;
   intCondition.Axis_28.Home.intout[0..9] := FALSE;
   intCondition.Axis_28.Jog.ForwardInterlockOK := FALSE;
   intCondition.Axis_28.Jog.BackwardInterlockOk := FALSE;
   intCondition.Axis_28.Jog.ForwardInterlockError := FALSE;
   intCondition.Axis_28.Jog.BackwardInterlockError := FALSE;
   intCondition.Axis_28.Jog.intOut[0..9] := FALSE;
   intCondition.Axis_28.Position.interlockOk[0..15] := FALSE;
   intCondition.Axis_28.Position.interlockError[0..15] := FALSE;
   intCondition.Axis_28.Position.intOut[0..9] := FALSE;
   intCondition.Axis_29.Home.HomeInterlock := FALSE;
   intCondition.Axis_29.Home.homeinterlock_error := FALSE;
   intCondition.Axis_29.Home.intout[0..9] := FALSE;
   intCondition.Axis_29.Jog.ForwardInterlockOK := FALSE;
   intCondition.Axis_29.Jog.BackwardInterlockOk := FALSE;
   intCondition.Axis_29.Jog.ForwardInterlockError := FALSE;
   intCondition.Axis_29.Jog.BackwardInterlockError := FALSE;
   intCondition.Axis_29.Jog.intOut[0..9] := FALSE;
   intCondition.Axis_29.Position.interlockOk[0..15] := FALSE;
   intCondition.Axis_29.Position.interlockError[0..15] := FALSE;
   intCondition.Axis_29.Position.intOut[0..9] := FALSE;
   intCondition.Axis_30.Home.HomeInterlock := FALSE;
   intCondition.Axis_30.Home.homeinterlock_error := FALSE;
   intCondition.Axis_30.Home.intout[0..9] := FALSE;
   intCondition.Axis_30.Jog.ForwardInterlockOK := FALSE;
   intCondition.Axis_30.Jog.BackwardInterlockOk := FALSE;
   intCondition.Axis_30.Jog.ForwardInterlockError := FALSE;
   intCondition.Axis_30.Jog.BackwardInterlockError := FALSE;
   intCondition.Axis_30.Jog.intOut[0..9] := FALSE;
   intCondition.Axis_30.Position.interlockOk[0..15] := FALSE;
   intCondition.Axis_30.Position.interlockError[0..15] := FALSE;
   intCondition.Axis_30.Position.intOut[0..9] := FALSE;
   intCondition.Axis_31.Home.HomeInterlock := FALSE;
   intCondition.Axis_31.Home.homeinterlock_error := FALSE;
   intCondition.Axis_31.Home.intout[0..9] := FALSE;
   intCondition.Axis_31.Jog.ForwardInterlockOK := FALSE;
   intCondition.Axis_31.Jog.BackwardInterlockOk := FALSE;
   intCondition.Axis_31.Jog.ForwardInterlockError := FALSE;
   intCondition.Axis_31.Jog.BackwardInterlockError := FALSE;
   intCondition.Axis_31.Jog.intOut[0..9] := FALSE;
   intCondition.Axis_31.Position.interlockOk[0..15] := FALSE;
   intCondition.Axis_31.Position.interlockError[0..15] := FALSE;
   intCondition.Axis_31.Position.intOut[0..9] := FALSE;
   intCondition.Axis_32.Home.HomeInterlock := FALSE;
   intCondition.Axis_32.Home.homeinterlock_error := FALSE;
   intCondition.Axis_32.Home.intout[0..9] := FALSE;
   intCondition.Axis_32.Jog.ForwardInterlockOK := FALSE;
   intCondition.Axis_32.Jog.BackwardInterlockOk := FALSE;
   intCondition.Axis_32.Jog.ForwardInterlockError := FALSE;
   intCondition.Axis_32.Jog.BackwardInterlockError := FALSE;
   intCondition.Axis_32.Jog.intOut[0..9] := FALSE;
   intCondition.Axis_32.Position.interlockOk[0..15] := FALSE;
   intCondition.Axis_32.Position.interlockError[0..15] := FALSE;
   intCondition.Axis_32.Position.intOut[0..9] := FALSE;
   intCondition.Axis_33.Home.HomeInterlock := FALSE;
   intCondition.Axis_33.Home.homeinterlock_error := FALSE;
   intCondition.Axis_33.Home.intout[0..9] := FALSE;
   intCondition.Axis_33.Jog.ForwardInterlockOK := FALSE;
   intCondition.Axis_33.Jog.BackwardInterlockOk := FALSE;
   intCondition.Axis_33.Jog.ForwardInterlockError := FALSE;
   intCondition.Axis_33.Jog.BackwardInterlockError := FALSE;
   intCondition.Axis_33.Jog.intOut[0..9] := FALSE;
   intCondition.Axis_33.Position.interlockOk[0..15] := FALSE;
   intCondition.Axis_33.Position.interlockError[0..15] := FALSE;
   intCondition.Axis_33.Position.intOut[0..9] := FALSE;
   intCondition.Actuator_33.Home_INT := FALSE;
   intCondition.Actuator_33.Work_INT := FALSE;
   intCondition.Actuator_33.Home_INT_Error := FALSE;
   intCondition.Actuator_33.Work_INT_Error := FALSE;
   intCondition.Actuator_33.intOut[0..9] := FALSE;
   intCondition.Actuator_34.Home_INT := FALSE;
   intCondition.Actuator_34.Work_INT := FALSE;
   intCondition.Actuator_34.Home_INT_Error := FALSE;
   intCondition.Actuator_34.Work_INT_Error := FALSE;
   intCondition.Actuator_34.intOut[0..9] := FALSE;
   intCondition.Actuator_35.Home_INT := FALSE;
   intCondition.Actuator_35.Work_INT := FALSE;
   intCondition.Actuator_35.Home_INT_Error := FALSE;
   intCondition.Actuator_35.Work_INT_Error := FALSE;
   intCondition.Actuator_35.intOut[0..9] := FALSE;
   intCondition.Actuator_36.Home_INT := FALSE;
   intCondition.Actuator_36.Work_INT := FALSE;
   intCondition.Actuator_36.Home_INT_Error := FALSE;
   intCondition.Actuator_36.Work_INT_Error := FALSE;
   intCondition.Actuator_36.intOut[0..9] := FALSE;
   intCondition.Actuator_37.Home_INT := FALSE;
   intCondition.Actuator_37.Work_INT := FALSE;
   intCondition.Actuator_37.Home_INT_Error := FALSE;
   intCondition.Actuator_37.Work_INT_Error := FALSE;
   intCondition.Actuator_37.intOut[0..9] := FALSE;
   intCondition.Actuator_38.Home_INT := FALSE;
   intCondition.Actuator_38.Work_INT := FALSE;
   intCondition.Actuator_38.Home_INT_Error := FALSE;
   intCondition.Actuator_38.Work_INT_Error := FALSE;
   intCondition.Actuator_38.intOut[0..9] := FALSE;
END_DATA_BLOCK
